FUNCTION_BLOCK FB_eChillerSystem EXTENDS FB_SystemContinous
VAR_INPUT
	fExternalTemperature : REAL; //External temperature of buffer storage
END_VAR
VAR_OUTPUT
END_VAR
VAR
	//Efficient Energy eChiller 45-II
	eChiller : FB_eChiller;
	
	//discrete valve 138
	ST_SV138DefaultParameters : ST_MixingValveDefaultParameters := (bFeedbackSignal := TRUE,aSetPointLimitsPosition := [0,100],fDefaultPosition := 0, aSetPointLimitsTemperature := [0,100], 
								fControllerAmplification := 0.265, tControllerIntegralTime := T#15S, 
								tTaskCycleTime := GlobalVariables.tTaskCycleTime, tCtrlCycleTime := T#5S);
	SV138 : FB_MixingValve := (ST_DefaultParameters := ST_SV138DefaultParameters); //valve motor needs continous signal but operates only between extreme positions	
	
	//internal variables
	bSetStatusOn_eChiller : BOOL;
	bSetStatusOn_SV138 : BOOL;
END_VAR

MAIN();
eChiller(
	bSetStatusOnAutomatic := bSetStatusOn_eChiller,
	fSetPointAutomatic := fSetPoint,
	bAlgorithmPermission := bAlgorithmPermission,
	fExternalTemperature := fExternalTemperature);
eChiller.SetState();

//valve may only control position, not temperatures
SV138(
	bSetStatusOnAutomatic := bSetStatusOn_SV138,
	fSetPointAutomatic := 100,
	bAlgorithmPermission := bAlgorithmPermission,
	nControlModeAutomatic := 0);
SV138.SetState_AI_AO();

METHOD PROTECTED  CheckError : BOOL
VAR_INPUT
END_VAR
VAR
	bError_eChiller : BOOL := FALSE;
	bError_SV138 : BOOL := FALSE;
END_VAR
VAR_OUTPUT
	bError : BOOL := FALSE;
END_VAR
//check chiller for error
bError_eChiller := eChiller.bError;

//check valve SV138 for error
IF SV138.fOperatingPoint <= 95 AND eChiller.bStatusOn THEN
	bError_SV138 := TRUE;
END_IF

bError := bError_eChiller OR bError_SV138;
END_METHOD

METHOD PROTECTED  Operational : BOOL
VAR_INPUT
END_VAR
VAR_OUTPUT
	bSwitchToWorking : BOOL := FALSE;
END_VAR
bSetStatusOn_eChiller := TRUE;

IF eChiller.bStatusOn THEN
	bSwitchToWorking := TRUE;
END_IF
END_METHOD

METHOD PROTECTED  RampDown : BOOL
VAR_INPUT
END_VAR
VAR_OUTPUT
	bRampDownFinished : BOOL := FALSE;
END_VAR
bSetStatusOn_eChiller := FALSE;

//wait until eChiller is switched off before closing valve
IF NOT eChiller.bStatusOn THEN
	bSetStatusOn_SV138 := FALSE;
END_IF

//wait until valve is closed and ensure that eChiller is not switched on meanwhile
IF SV138.fOperatingPoint < 5 AND NOT eChiller.bStatusOn THEN
	bRampDownFinished := TRUE;
END_IF
END_METHOD

METHOD PROTECTED  RampUp : BOOL
VAR_INPUT
END_VAR
VAR_OUTPUT
	bRampUpFinished : BOOL := FALSE;
END_VAR
bSetStatusOn_SV138 := TRUE;

//wait until valve is opened
IF SV138.fOperatingPoint > 95 THEN
	bRampUpFinished := TRUE;
END_IF
END_METHOD

METHOD PROTECTED   SetSetPointLimits : BOOL
VAR_INPUT
END_VAR
aSetPointLimits[1] := eChiller.ST_DefaultParameters.aSetPointLimitsTemperature[1];
aSetPointLimits[2] := eChiller.ST_DefaultParameters.aSetPointLimitsTemperature[2];
END_METHOD

METHOD PROTECTED  Working : BOOL
VAR_INPUT
END_VAR
VAR_OUTPUT
	bSwitchToOperational : BOOL := FALSE;
END_VAR
//check if eChiller is switched off (manually) but valve is still opened
END_METHOD

END_FUNCTION_BLOCK

(* stored: Version 1.1.0.1, ProductVersion 3.1.4024.10
   POU FB_eChillerSystem: Id {761e262d-2727-4279-88a1-3ac73010bbca}, SpecialFunc None
   Method CheckError: Id {87b68d69-7506-4fd5-920f-31c8ac6bc4f2}
   Method Operational: Id {830bd434-77f6-4d32-9616-294163c3dc90}
   Method RampDown: Id {e920d523-a5e9-4cce-a828-b16d80d8611f}
   Method RampUp: Id {a35d72c4-c137-4825-b9db-822abc1571be}
   Method SetSetPointLimits: Id {a4e2465f-3e29-44c1-a39b-c5d763bbb0bc}
   Method Working: Id {40c6e2d0-ac93-45e6-921b-d845a8bf1ef9} *)
